{attribute 'qualified_only'}
VAR_GLOBAL
	nTime_multiplier:		INT:=1;
	nSeconds:				INT;
	nMinutes:				INT;
	nHours:					INT;
	nCycle:					INT;
	nMontakohalvinta:		INT(1..95):=20;
	nMontakokalleinta:		INT(1..95):=20;
	nHintaRajaPumppaus:		REAL :=3.0;
	nHintaRajaTuotanto:		REAL :=7.0;
	fprice:					REAL;
	
	// DUT:eissa määriteltiin mitä tietoja structit sisältää. Tässä tehdään muuttuja structissa, jossa tieto asuu. yhdistetään HMI:hin
	stEsimerkki				: ST_Esimerkki;
	
	stGenerator				: ST_GeneratorHmi;
	// Laitoin genun GVL:ään -> helppo työntää rajapinnan kautta tietoja esim roomtempille.
	fbGenerator				: FB_Generator;
	
	stRoomTemp				: ST_RoomTempHmi;
	fbRoomtemp				: FB_RoomTemp;
END_VAR

(* stored: Version 1.1.0.1
   GVL GVL: Id {4525eb99-dc14-4c5d-a458-25eeb85211f8} *)
